// TIA Portal V20 export
DATA_BLOCK "InstGetAxisStatus"   // DB2
AUTHOR : Siemens Digital Industries
FAMILY : LAF
NAME : LAF_GetAxisStatus
VERSION : 1.1
// stored: InstanceOfName LAF_GetAxisStatus, InstanceOfType FB
"LAF_GetAxisStatus"
   // VAR_INPUT
   //    enable : Bool := TRUE;
   // END_VAR
   // VAR_OUTPUT
   //    valid { ExternalWritable := 'False'} : Bool := FALSE;
   //    busy { ExternalWritable := 'False'} : Bool := FALSE;
   //    error { ExternalWritable := 'False'} : Bool := FALSE;
   //    status { ExternalWritable := 'False'} : Word := 16#7000;
   //    diagnostics { ExternalWritable := 'False'} : "LAF_typeDiagnostics";
   // END_VAR
   // VAR_IN_OUT
   //    configuration : Array[*] of "LAF_typeDriveDiagConfig";
   //    moduleInterface : "LAF_typeDriveDiagInterfaceHmi";
   // END_VAR
   // VAR
   //    statInternal { ExternalAccessible := 'False'; ExternalVisible := 'False'; ExternalWritable := 'False'} : Struct
   //       enablePrevious : Bool := FALSE;
   //       valid : Bool := FALSE;
   //       busy : Bool := FALSE;
   //       error : Bool := FALSE;
   //       errorUserCleared : Bool := FALSE;
   //       errorAutoCleared : Bool := FALSE;
   //       disablingCompleted : Bool := TRUE;
   //       diagnostics : "LAF_typeDiagnostics";
   //       emptyDiagnostics : "LAF_typeDiagnostics";
   //    END_STRUCT;
   //    statMainState { ExternalAccessible := 'False'; ExternalVisible := 'False'; ExternalWritable := 'False'} : DInt := 0;
   //    statArrayMin { ExternalAccessible := 'False'; ExternalVisible := 'False'; ExternalWritable := 'False'} : DInt := 0;
   //    statArrayMax { ExternalAccessible := 'False'; ExternalVisible := 'False'; ExternalWritable := 'False'} : DInt := 41;
   // END_VAR
BEGIN
   diagnostics.status := 16#7000;
   diagnostics.subfunctionStatus := 16#0000;
   diagnostics.stateNumber := 0;
   statInternal.diagnostics.status := 16#7000;
   statInternal.diagnostics.subfunctionStatus := 16#0000;
   statInternal.diagnostics.stateNumber := 50;
   statInternal.emptyDiagnostics.status := 16#7000;
   statInternal.emptyDiagnostics.subfunctionStatus := 16#0000;
   statInternal.emptyDiagnostics.stateNumber := 0;
END_DATA_BLOCK
